FUNCTION F_SimpleDeadBand : BOOL
VAR_INPUT
	rActualValue:REAL;		(*Actual Value measured*)
	rTolerance:REAL;			(*measurement Tolerance*)
	rReferenceValue:REAL;	(*Reference value*)
END_VAR
VAR
END_VAR

(*Dead Band calculation according to the given parameters*)
F_SimpleDeadBand:= betwenLimits(rReferenceValue-rTolerance, rActualValue, rReferenceValue+rTolerance);

END_FUNCTION

(* stored: Version 1.1.0.1, ProductVersion 3.1.4024.12
   POU F_SimpleDeadBand: Id {1a4d07d9-f46a-4d88-80f8-8a8c204e9610}, SpecialFunc None *)
